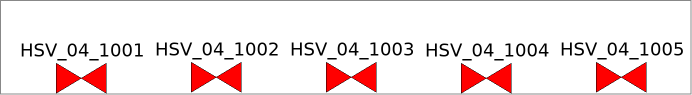
VISUALIZATION Visualization  // 692x95
    Group (15,24 135x69)
        OnMouseClick: OpenDialog Dialog=HSV_04_1001, OpenModal=True, OpenCentered=True
        Polygon (41,39) (41,69) (66,54), invisible if: NOT progHSVCntrl.HSV_04_1001.FB_Close
        Polygon (91,39) (91,69) (66,54), invisible if: NOT progHSVCntrl.HSV_04_1001.FB_Close
        Polygon (41,39) (41,69) (66,54), invisible if: NOT progHSVCntrl.HSV_04_1001.FB_Travelling
        Polygon (91,39) (91,69) (66,54), invisible if: NOT progHSVCntrl.HSV_04_1001.FB_Travelling
        Polygon (41,39) (41,69) (66,54), invisible if: NOT progHSVCntrl.HSV_04_1001.FB_Open
        Polygon (91,39) (91,69) (66,54), invisible if: NOT progHSVCntrl.HSV_04_1001.FB_Open
        Polygon (41,39) (41,69) (66,54), invisible if: NOT progHSVCntrl.HSV_04_1001.Alarm
        Polygon (91,39) (91,69) (66,54), invisible if: NOT progHSVCntrl.HSV_04_1001.Alarm
        Label (0,0 135x53), "HSV_04_1001"
    Group (150,23 135x69)
        OnMouseClick: OpenDialog Dialog=HSV_04_1002, OpenModal=True, OpenCentered=True
        Polygon (41,39) (41,69) (66,54), invisible if: NOT progHSVCntrl.HSV_04_1002.FB_Close
        Polygon (91,39) (91,69) (66,54), invisible if: NOT progHSVCntrl.HSV_04_1002.FB_Close
        Polygon (41,39) (41,69) (66,54), invisible if: NOT progHSVCntrl.HSV_04_1002.FB_Travelling
        Polygon (91,39) (91,69) (66,54), invisible if: NOT progHSVCntrl.HSV_04_1002.FB_Travelling
        Polygon (41,39) (41,69) (66,54), invisible if: NOT progHSVCntrl.HSV_04_1002.FB_Open
        Polygon (91,39) (91,69) (66,54), invisible if: NOT progHSVCntrl.HSV_04_1002.FB_Open
        Polygon (41,39) (41,69) (66,54), invisible if: NOT progHSVCntrl.HSV_04_1002.Alarm
        Polygon (91,39) (91,69) (66,54), invisible if: NOT progHSVCntrl.HSV_04_1002.Alarm
        Label (0,0 135x53), "HSV_04_1002"
    Group (285,23 135x69)
        OnMouseClick: OpenDialog Dialog=HSV_04_1003, OpenModal=True, OpenCentered=True
        Polygon (41,39) (41,69) (66,54), invisible if: NOT progHSVCntrl.HSV_04_1003.FB_Close
        Polygon (91,39) (91,69) (66,54), invisible if: NOT progHSVCntrl.HSV_04_1003.FB_Close
        Polygon (41,39) (41,69) (66,54), invisible if: NOT progHSVCntrl.HSV_04_1003.FB_Travelling
        Polygon (91,39) (91,69) (66,54), invisible if: NOT progHSVCntrl.HSV_04_1003.FB_Travelling
        Polygon (41,39) (41,69) (66,54), invisible if: NOT progHSVCntrl.HSV_04_1003.FB_Open
        Polygon (91,39) (91,69) (66,54), invisible if: NOT progHSVCntrl.HSV_04_1003.FB_Open
        Polygon (41,39) (41,69) (66,54), invisible if: NOT progHSVCntrl.HSV_04_1003.Alarm
        Polygon (91,39) (91,69) (66,54), invisible if: NOT progHSVCntrl.HSV_04_1003.Alarm
        Label (0,0 135x53), "HSV_04_1003"
    Group (420,24 135x69)
        OnMouseClick: OpenDialog Dialog=HSV_04_1004, OpenModal=True, OpenCentered=True
        Polygon (41,39) (41,69) (66,54), invisible if: NOT progHSVCntrl.HSV_04_1004.FB_Close
        Polygon (91,39) (91,69) (66,54), invisible if: NOT progHSVCntrl.HSV_04_1004.FB_Close
        Polygon (41,39) (41,69) (66,54), invisible if: NOT progHSVCntrl.HSV_04_1004.FB_Travelling
        Polygon (91,39) (91,69) (66,54), invisible if: NOT progHSVCntrl.HSV_04_1004.FB_Travelling
        Polygon (41,39) (41,69) (66,54), invisible if: NOT progHSVCntrl.HSV_04_1004.FB_Open
        Polygon (91,39) (91,69) (66,54), invisible if: NOT progHSVCntrl.HSV_04_1004.FB_Open
        Polygon (41,39) (41,69) (66,54), invisible if: NOT progHSVCntrl.HSV_04_1004.Alarm
        Polygon (91,39) (91,69) (66,54), invisible if: NOT progHSVCntrl.HSV_04_1004.Alarm
        Label (0,0 135x53), "HSV_04_1004"
    Group (555,23 135x69)
        Polygon (41,39) (41,69) (66,54), invisible if: NOT progHSVCntrl.HSV_04_1005.FB_Close
        Polygon (91,39) (91,69) (66,54), invisible if: NOT progHSVCntrl.HSV_04_1005.FB_Close
        Polygon (41,39) (41,69) (66,54), invisible if: NOT progHSVCntrl.HSV_04_1005.FB_Travelling
        Polygon (91,39) (91,69) (66,54), invisible if: NOT progHSVCntrl.HSV_04_1005.FB_Travelling
        Polygon (41,39) (41,69) (66,54), invisible if: NOT progHSVCntrl.HSV_04_1005.FB_Open
        Polygon (91,39) (91,69) (66,54), invisible if: NOT progHSVCntrl.HSV_04_1005.FB_Open
        Polygon (41,39) (41,69) (66,54), invisible if: NOT progHSVCntrl.HSV_04_1005.Alarm
        Polygon (91,39) (91,69) (66,54), invisible if: NOT progHSVCntrl.HSV_04_1005.Alarm
        Label (0,0 135x53), "HSV_04_1005"
END_VISUALIZATION

(* stored: Version 1.1.0.1, ProductVersion 3.1.4022.17
   Visu Visualization: Id {7958c93a-f917-4dba-ba1d-3675467214dc} *)
